Fanuc KAREL source: kt00923.KL

-- PROVISIONAL review KL for V1013-1; original PC SHA256 0ffc9f9f81182c2b2ef81ad5b4a842c7258e9706fb54423a6bceac36350e4bc9
-- Incomplete behavior may be omitted. Consult companion uncertainty JSON. Do not deploy.
PROGRAM KT00923
%NOLOCKGROUP
VAR
  S1 : STRING[80]
  S2 : STRING[80]
  OUT : STRING[80]
BEGIN
  -- UNRESOLVED_PC offsets 5-14; opcodes 3F,75
  -- UNRESOLVED_PC offsets 19-28; opcodes 3F,75
  -- UNRESOLVED_PC offsets 33-42; opcodes 3F,75
  -- UNRESOLVED_PC offsets 47-56; opcodes 3F,75
  -- UNRESOLVED_PC offsets 61-82; opcodes 27,22,2A,27,9D,27,9D,76,75
  -- UNRESOLVED_PC offsets 87-91; opcodes 7F
END KT00923
